FUNCTION_BLOCK AR_model
  (* Version 1.0, 2005-09-21, Goran Cengic, Chalmers *)
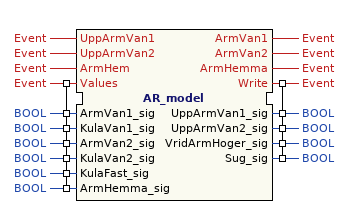
  EVENT_INPUT
    UppArmVan1;
    UppArmVan2;
    ArmHem;
    Values WITH ArmVan1_sig, KulaVan1_sig, ArmVan2_sig, KulaVan2_sig, KulaFast_sig, ArmHemma_sig;
  END_EVENT
  EVENT_OUTPUT
    ArmVan1;
    ArmVan2;
    ArmHemma;
    Write WITH UppArmVan1_sig, UppArmVan2_sig, VridArmHoger_sig, Sug_sig;
  END_EVENT
  VAR_INPUT
    ArmVan1_sig : BOOL;
    KulaVan1_sig : BOOL;
    ArmVan2_sig : BOOL;
    KulaVan2_sig : BOOL;
    KulaFast_sig : BOOL;
    ArmHemma_sig : BOOL;
  END_VAR
  VAR_OUTPUT
    UppArmVan1_sig : BOOL;
    UppArmVan2_sig : BOOL;
    VridArmHoger_sig : BOOL;
    Sug_sig : BOOL;
  END_VAR
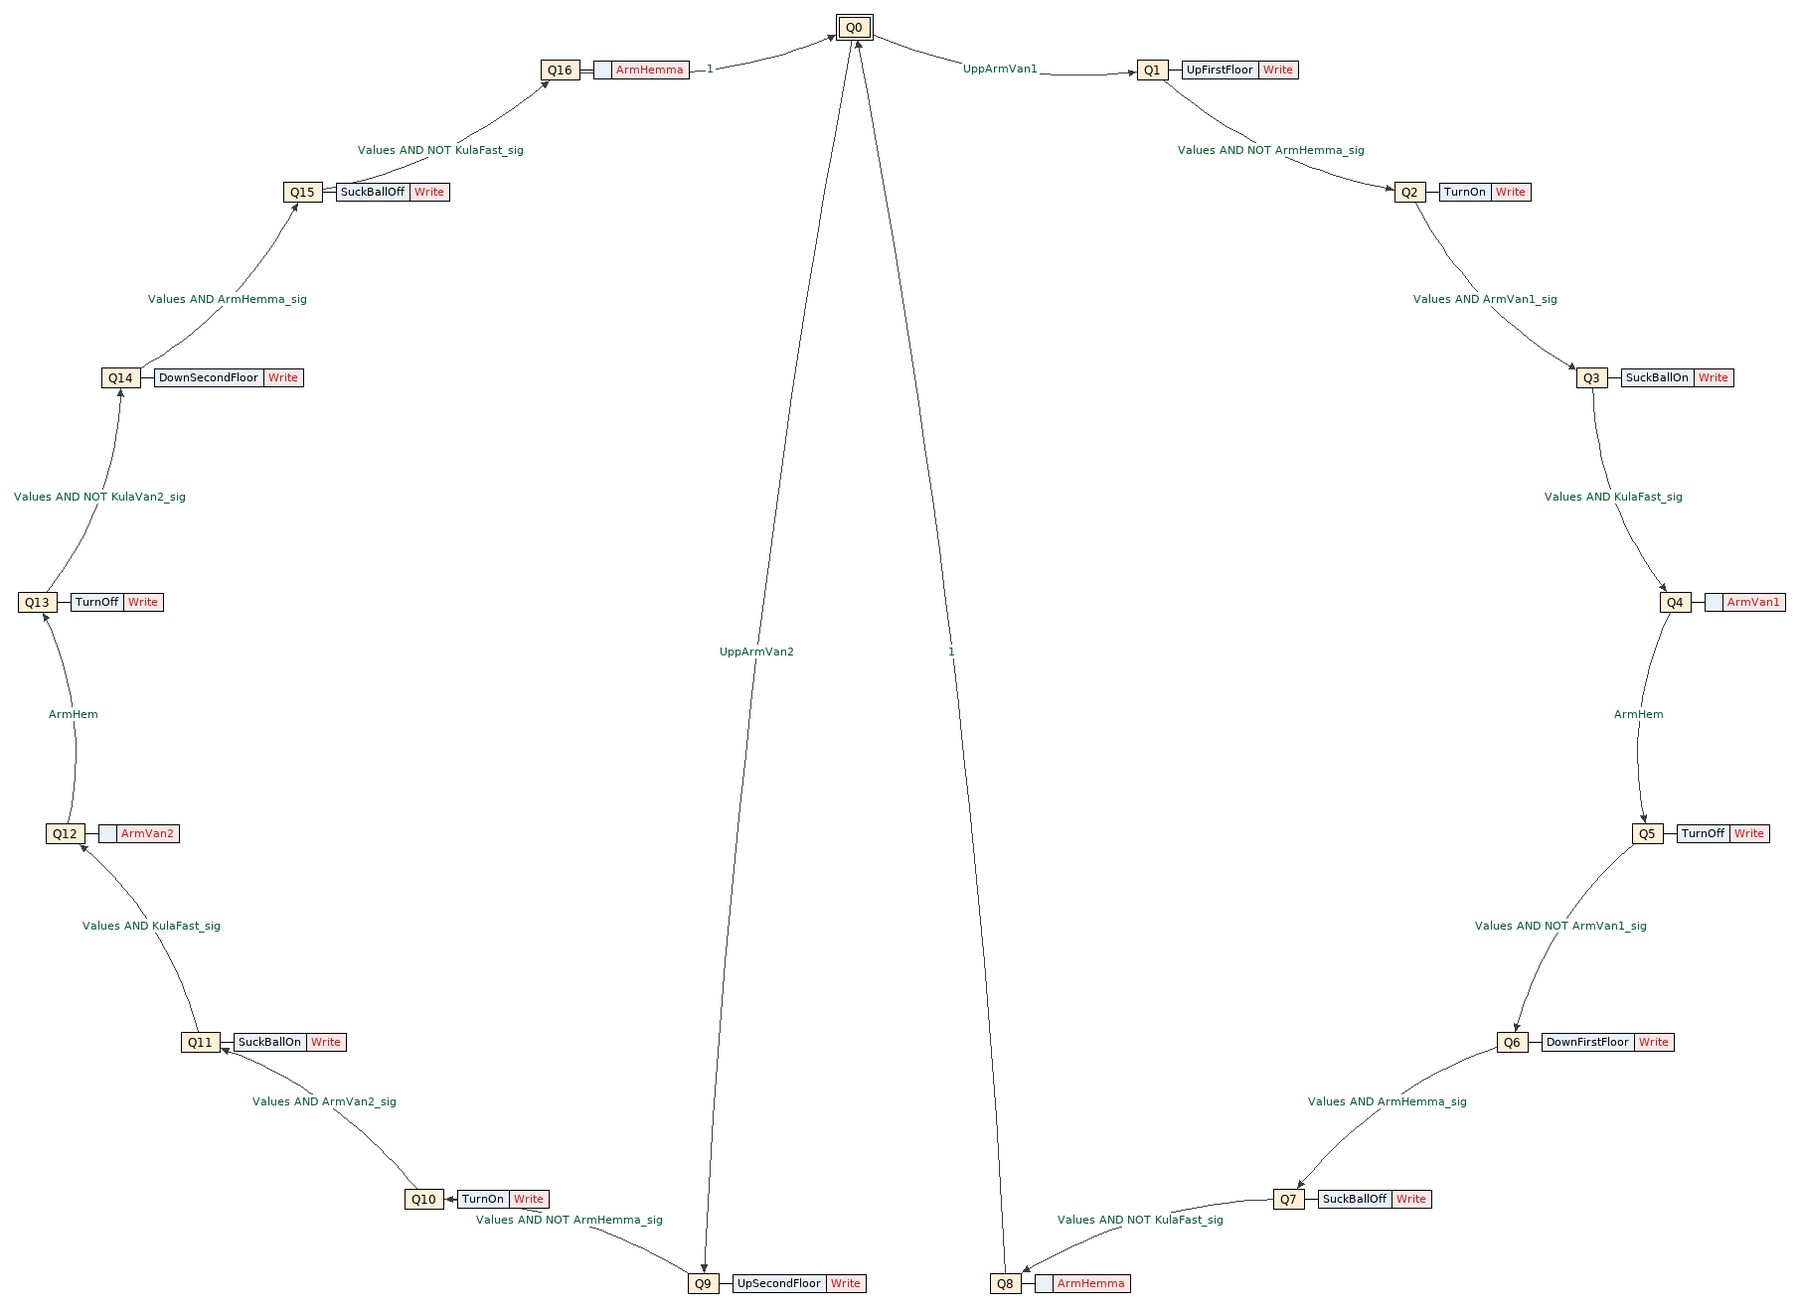
  EC_STATES
    Q0;
    Q1 : UpFirstFloor -> Write;
    Q2 : TurnOn -> Write;
    Q3 : SuckBallOn -> Write;
    Q4 : -> ArmVan1;
    Q5 : TurnOff -> Write;
    Q6 : DownFirstFloor -> Write;
    Q7 : SuckBallOff -> Write;
    Q8 : -> ArmHemma;
    Q9 : UpSecondFloor -> Write;
    Q10 : TurnOn -> Write;
    Q11 : SuckBallOn -> Write;
    Q12 : -> ArmVan2;
    Q13 : TurnOff -> Write;
    Q14 : DownSecondFloor -> Write;
    Q15 : SuckBallOff -> Write;
    Q16 : -> ArmHemma;
  END_STATES
  EC_TRANSITIONS
    Q0 TO Q1 := UppArmVan1;
    Q1 TO Q2 := Values AND NOT ArmHemma_sig;
    Q2 TO Q3 := Values AND ArmVan1_sig;
    Q3 TO Q4 := Values AND KulaFast_sig;
    Q4 TO Q5 := ArmHem;
    Q5 TO Q6 := Values AND NOT ArmVan1_sig;
    Q6 TO Q7 := Values AND ArmHemma_sig;
    Q7 TO Q8 := Values AND NOT KulaFast_sig;
    Q8 TO Q0 := 1;
    Q0 TO Q9 := UppArmVan2;
    Q9 TO Q10 := Values AND NOT ArmHemma_sig;
    Q10 TO Q11 := Values AND ArmVan2_sig;
    Q11 TO Q12 := Values AND KulaFast_sig;
    Q12 TO Q13 := ArmHem;
    Q13 TO Q14 := Values AND NOT KulaVan2_sig;
    Q14 TO Q15 := Values AND ArmHemma_sig;
    Q15 TO Q16 := Values AND NOT KulaFast_sig;
    Q16 TO Q0 := 1;
  END_TRANSITIONS
  ALGORITHM TurnOn IN Java:
		System.out.println("Arm turning right.");
		VridArmHoger_sig = true;
  END_ALGORITHM
  ALGORITHM TurnOff IN Java:
		System.out.println("Arm turning left.");
		VridArmHoger_sig = false;
  END_ALGORITHM
  ALGORITHM SuckBallOn IN Java:
		System.out.println("Arm sucking ball.");
		Sug_sig = true;
  END_ALGORITHM
  ALGORITHM SuckBallOff IN Java:
		System.out.println("Arm releasing ball.");
		Sug_sig = false;
  END_ALGORITHM
  ALGORITHM UpSecondFloor IN Java:
		System.out.println("Arm going up to second floor.");
		UppArmVan1_sig = true;
		UppArmVan2_sig = true;
  END_ALGORITHM
  ALGORITHM DownSecondFloor IN Java:
		System.out.println("Arm going down from second floor.");
		UppArmVan1_sig = false;
		UppArmVan2_sig = false;
  END_ALGORITHM
  ALGORITHM UpFirstFloor IN Java:
		System.out.println("Arm going up to first floor.");
		UppArmVan1_sig = true;
  END_ALGORITHM
  ALGORITHM DownFirstFloor IN Java:
		System.out.println("Arm going down from first floor.");
		UppArmVan1_sig = false;
  END_ALGORITHM
END_FUNCTION_BLOCK
